Staubli VAL3: setAllAccel.pgx

public program setAllAccel(num x_nNewValue (dimensions=1), num x_nOldValue (dimensions=1))
  local num i
  local num l_nSize
  local TrajectoryItem l_tTraj
begin
  //
  // change all the accel(equal at newValue)to the newValue
  //
  if x_nNewValue!=x_nOldValue
    call trajType:getSizeItem(false,l_nSize)
    // scan it
    for i=0 to (l_nSize-1)
      // get it
      call trajType:getTrajItem(l_tTraj,i)
      // check if is OK
      if l_tTraj.nom_speed.accel==x_nOldValue
        l_tTraj.nom_speed.accel=l_tTraj.nom_speed.decel=x_nNewValue
      endIf
      // set IT
      call trajType:setTrajItem(l_tTraj,i)
    endFor
  endIf
end
